FUNCTION_BLOCK FB_BufferStorage
VAR_INPUT
END_VAR
VAR_OUTPUT
	UpperTemperature : REAL;
	MidTemperature : REAL;
	LowerTemperature : REAL;
END_VAR
VAR
	UpperTemperatureSensor : FB_TemperatureSensor; //upper temperature sensor
	MidTemperatureSensor : FB_TemperatureSensor; //mid temperature sensor
	LowerTemperatureSensor : FB_TemperatureSensor; //lower temperature sensor
END_VAR

//get sensor inputs
UpperTemperatureSensor.SetState_AI();
MidTemperatureSensor.SetState_AI();
LowerTemperatureSensor.SetState_AI();

//Set outputs
UpperTemperature := UpperTemperatureSensor.fTemperature;
MidTemperature := MidTemperatureSensor.fTemperature;
LowerTemperature := LowerTemperatureSensor.fTemperature;

END_FUNCTION_BLOCK

(* stored: Version 1.1.0.1, ProductVersion 3.1.4024.9
   POU FB_BufferStorage: Id {8e38393d-195d-45df-94d3-1eb118fb470f}, SpecialFunc None *)
